TEXTLIST ErrorList
  0 = 'no error' | de: 'kein Fehler' | fr: 'pas de Erreur'
  100 = 'Actuator | Autorisation refused for action Go Out' | de: 'Aktor | Keine Autorisation zum ausfahren' | fr: 'Actionneur | Pas de autorisation pour étendre'
  101 = 'Actuator | Autorisation refused for action Go In' | de: 'Aktor | Keine Autorisation zum einfahren' | fr: 'Actionneur | Pas de autorisation pour retracter'
  110 = 'Actuator | Error timeout go-out' | de: 'Aktor | Timeout ausfahren' | fr: 'Actionneur | Timeout  étendre'
  111 = 'Actuator | Error timeout go-in' | de: 'Aktor | Timeout einfahren' | fr: 'Actionneur | Timeout retracter'
  120 = 'Actuator | Both sensors (IxSensIn & IxSensOut) at the same time' | de: 'Aktor | Beide Sensoren sind gleichzeitig aktiv' | fr: 'Actionneur | Les deux capteurs sont vrai en meme temps'
  121 = 'Actuator | Where shall I go? xSetSort=1 et xSetRentre=1' | de: 'Aktor | Was soll ich tun? xSetSort=1 und xSetRentre=1' | fr: 'Actionneur | Sortir ou rentrer? xSetSort=1 et xSetRentre=1'
  200 = 'Auto | Vision | Error while detecting original object' | de: 'Auto | Vision | Fehler beim Erkennen des Start-Objektes' | fr: "Auto | Vision | Erreur detecter l'object de départ"
  210 = 'Auto | Timeout - Motor did not reach desired speed' | de: 'Auto | Timeout - Motor hat nicht schnell genug den Soll-Wert erreicht' | fr: 'Auto | Timeout - Moteur a pas atteint la vitesse de consigne assez rapide'
  201 = 'Auto | Vision | Error detecting processed object' | de: 'Auto | Vision | Fehler beim Erkennen des End-Objektes' | fr: 'Auto | Vision | Erreur detecter object de fin'
  300 = 'fbMotor | Error in PID-Loop' | de: 'fbMotor | Fehler in der PID-Schleife' | fr: 'fbMotor | Erreur dans boucle PID'
  301 = 'fbMotor | Unable to reach Setpoint Speed' | de: 'fbMotor | Kann Setpoint-Wert nicht erreichen' | fr: "fbMoteur | Impossible d'atteindre la vitesse de consigne"
  401 = 'fbTCP | mReceive | Received Data was lost' | de: 'fbTCP | mReceive | Verlust von eingehenden Daten ' | fr: 'fbTCP | mReceive | Perte de donnes en entree'
  402 = 'fbTCP | Error sending data' | de: 'fbTCP | Fehler beim Senden der Daten' | fr: "fbTCP | Probleme lorsque de l'envoi des données"
  403 = 'fbTCP | Error connecting /disconnecting to Server' | de: 'fbTCP | Fehler beim Verbinden / Trennen der Verbindung zum Server' | fr: 'fbTCP | Erreur lorsque de la (de-)connexion aux Serveur'
  404 = 'fbTCP | mReceive | Error while Receiving data' | de: 'fbTCP | mReceive | Fehler beim Empfangen von Daten' | fr: 'fbTCP | mReceive | Probleme de réception'
  202 = 'Auto | Camera | Error while taking image'
  1 = 'Air Pressure low' | de: 'Luftdruck zu gering' | fr: "Pression d'air trop basse"
   = ''
END_TEXTLIST

(* stored: Version 1.1.0.1, ProductVersion 3.1.4020.6
   TextList ErrorList: Id {fbbf4080-7032-4e41-87a0-9d3e8bd94934} *)
